FUNCTION_BLOCK ZONE_VIEWL (* HVAC Zone View with Local Data Publish/Subscribe *)
  (* Standard: 61499-1; ApplicationDomain: HVAC; Function: View *)
  (* Version 0.0, 2006-04-07, JHC, Holobloc Inc *)
  (* Compiler header: package fb.rt.hvac; import fb.rt.net.*; import fb.rt.mva.*; *)
  (* Compiler classdef: public class ZONE_VIEWL extends FBMVCD *)
  (* Compiler Java Sun JDK 1.5.0 *)
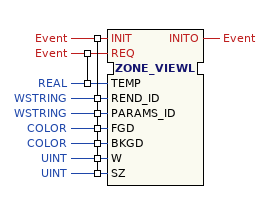
  EVENT_INPUT
    INIT WITH REND_ID, PARAMS_ID, BKGD, FGD, W, SZ; (* Initialize *)
    REQ WITH TEMP; (* TEMP display request *)
  END_EVENT
  EVENT_OUTPUT
    INITO; (* Initialized *)
  END_EVENT
  VAR_INPUT
    TEMP : REAL; (* Room Temperature, deg. F *)
    REND_ID : WSTRING; (* TEMP, FLOW subscriber channel ID *)
    PARAMS_ID : WSTRING := "PARAMS"; (* STEMP, XTEMP, LOAD subscriber channel ID *)
    FGD : COLOR := COLOR#white; (* Foreground Color *)
    BKGD : COLOR := COLOR#blue; (* Background Color *)
    W : UINT; (* Square room side dimension in pixels *)
    SZ : UINT := 12; (* Font size in points *)
  END_VAR
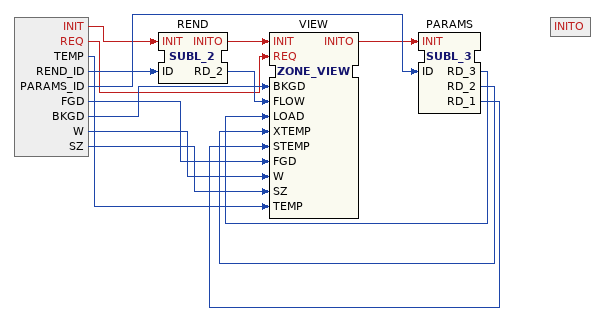
  FBS
    REND : SUBL_2;
    VIEW : ZONE_VIEW;
    PARAMS : SUBL_3;
  END_FBS
  EVENT_CONNECTIONS
    INIT TO REND.INIT;
    REND.INITO TO VIEW.INIT;
    VIEW.INITO TO PARAMS.INIT;
    REQ TO VIEW.REQ;
  END_CONNECTIONS
  DATA_CONNECTIONS
    REND_ID TO REND.ID;
    BKGD TO VIEW.BKGD;
    REND.RD_2 TO VIEW.FLOW;
    PARAMS_ID TO PARAMS.ID;
    PARAMS.RD_3 TO VIEW.LOAD;
    PARAMS.RD_2 TO VIEW.XTEMP;
    PARAMS.RD_1 TO VIEW.STEMP;
    FGD TO VIEW.FGD;
    W TO VIEW.W;
    SZ TO VIEW.SZ;
    TEMP TO VIEW.TEMP;
  END_CONNECTIONS
END_FUNCTION_BLOCK
